% RSLogix 500 project ALARMA.RSS, saved by version 8.40.00.08 %
PROJECT "ALARMA"    % processor: MicroLogix 1500 %

PROGRAM FILES
  LAD 2   4 rungs

DATA FILES
  O0 OUTPUT  4 elements
  I1 INPUT  6 elements
  S2 STATUS  66 elements
  B3 BINARY  1 elements
  T4 TIMER  1 elements
  C5 COUNTER  1 elements
  R6 CONTROL  1 elements
  N7 INTEGER  1 elements
  F8 FLOAT  1 elements

LADDER 2
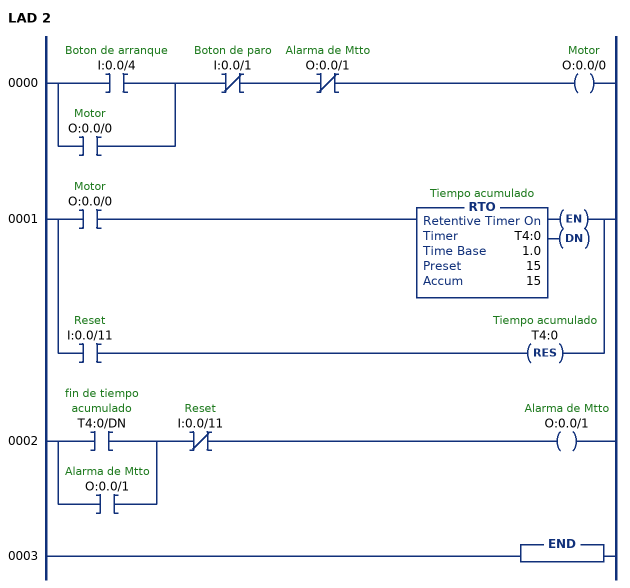
% Rung: 0 %
SOR BST XIC I:0.0/4 NXB XIC O:0.0/0 BND XIO I:0.0/1 XIO O:0.0/1 OTE O:0.0/0 EOR
%   I:0.0/4  "Boton de arranque" %
%   O:0.0/0  "Motor" %
%   I:0.0/1  "Boton de paro" %
%   O:0.0/1  "Alarma de Mtto" %
% Rung: 1 %
SOR BST XIC O:0.0/0 RTO T4:0 1.0 15 15 NXB XIC I:0.0/11 RES T4:0 BND EOR
%   O:0.0/0  "Motor" %
%   T4:0  "Tiempo acumulado" %
%   I:0.0/11  "Reset" %
% Rung: 2 %
SOR BST XIC T4:0/DN NXB XIC O:0.0/1 BND XIO I:0.0/11 OTE O:0.0/1 EOR
%   T4:0/DN  "fin de tiempo acumulado" %
%   O:0.0/1  "Alarma de Mtto" %
%   I:0.0/11  "Reset" %
% Rung: 3 %
SOR END EOR

DATA TABLE (non-zero values as saved)
DATA T4
% .PRE .ACC %
% T4:0 % 15 15
